FUNCTION_BLOCK FB_Station IMPLEMENTS IStation
VAR_INPUT
END_VAR
VAR_OUTPUT
END_VAR
VAR
    _Position          : REFERENCE TO FB_Position;
    _Process           : REFERENCE TO FB_AUT_ABSTRACT;
    _WaitPosOffset     : LREAL; // offset of the station position, should always be negative
    _iMaxWaitingMovers : INT;   // Maximum of waiting mover in front of the station

    _ApproachScenario : ApproachScenario_e := ApproachScenario_e.WaitOnFinishedProcess;

    _iID : INT := 0; // instance ID, is set during FB_Init using the value of _iInstanceCounter 
END_VAR
VAR_STAT
    _iInstanceCounter : INT := 1; // instance counter
END_VAR

PROPERTY ApproachScenario : ApproachScenario_e
GET
ApproachScenario := THIS^._ApproachScenario;
END_GET
SET
THIS^._ApproachScenario := ApproachScenario;
END_SET
END_PROPERTY

// Return true if the given object is equal to THIS^
METHOD Equals : BOOL
VAR_INPUT
    Station : REFERENCE TO FB_Station;
END_VAR
Equals := FALSE;

IF __ISVALIDREF(Station) THEN
    Equals := THIS = ADR(Station);
END_IF
END_METHOD

METHOD FB_init : BOOL
VAR_INPUT
    bInitRetains      : BOOL; // if TRUE, the retain variables are initialized (warm start / cold start)
    bInCopyCode       : BOOL; // if TRUE, the instance afterwards gets moved into the copy code (online change)
    Position          : REFERENCE TO FB_Position;
    Process           : REFERENCE TO FB_AUT_ABSTRACT;
    WaitPosOffset     : LREAL;
    ApproachScenario  : ApproachScenario_e;
    iMaxWaitingMovers : INT;
END_VAR
THIS^._iID               := THIS^._iInstanceCounter;
THIS^._iInstanceCounter  := THIS^._iInstanceCounter + 1;
THIS^._Position          REF= Position;
THIS^._Process           REF= Process;
THIS^._WaitPosOffset     := WaitPosOffset;
THIS^._ApproachScenario  := ApproachScenario;
THIS^._iMaxWaitingMovers := iMaxWaitingMovers;
END_METHOD

// the maxuimum number of waiting movers at the front of the station
PROPERTY iMaxWaitingMovers : INT
GET
iMaxWaitingMovers := THIS^._iMaxWaitingMovers;
END_GET
SET
THIS^._iMaxWaitingMovers := iMaxWaitingMovers;
END_SET
END_PROPERTY

PROPERTY Position : REFERENCE TO FB_Position
GET
Position REF=_Position;
END_GET
SET
_Position REF=Position;
END_SET
END_PROPERTY

PROPERTY Process : REFERENCE TO FB_AUT_ABSTRACT
GET
Process REF=_Process;
END_GET
SET
_Process REF= Process;
END_SET
END_PROPERTY

METHOD SetWaitPosOffset : REFERENCE TO FB_Station
VAR_INPUT
	WaitPosOffset : LREAL; // offset position from the given station, must be negative
END_VAR
IF _WaitPosOffset < 0 THEN
    _WaitPosOffset := WaitPos;
END_IF

SetWaitPosOffset REF= THIS^;
END_METHOD

METHOD ToString : STRING
VAR_INPUT
END_VAR
VAR
END_VAR
ToString := CONCAT('FB_Station_', TO_STRING(THIS^._iID));
END_METHOD

PROPERTY PUBLIC WaitPos : LREAL
GET
WaitPos := _WaitPosOffset + this^._Position.lrWorkPosition;
END_GET
SET
IF WaitPos < THIS^._Position.lrWorkPosition THEN
    _WaitPosOffset := WaitPos - THIS^._Position.lrWorkPosition;
END_IF
END_SET
END_PROPERTY

END_FUNCTION_BLOCK

(* stored: Version 1.1.0.1, ProductVersion 3.1.4024.6
   POU FB_Station: Id {76f3a0a5-7330-41a9-8dcd-67e3fa45891a}, SpecialFunc None
   Property ApproachScenario: Id {39b39f49-19c1-4773-90ff-7d9f9dd0bc2b}
   Get Get: Id {c7ab1366-26ac-4d26-8a07-2e23989dbdf5}
   Set Set: Id {c657ec57-92e0-4d09-9356-1fe7958f2743}
   Method Equals: Id {c76b8ece-aab6-47d5-90c3-9d4c81b08fdb}
   Method FB_init: Id {898dafd4-0828-4ee9-bb08-7822f297b3cc}
   Property iMaxWaitingMovers: Id {6a45a41f-3689-4688-9ba9-b8da1a5ddf71}
   Get Get: Id {e9a9e870-7f1d-4040-b314-a5cfa5de9a7d}
   Set Set: Id {15534dbf-4933-48be-bdb5-55a0a0a3d73e}
   Property Position: Id {b021e593-80f7-4dca-adcc-e8a0edd62ea6}
   Get Get: Id {4a41f306-d439-4214-a524-8ce6f093a989}
   Set Set: Id {062b4c53-3279-46a7-994d-891e38993d44}
   Property Process: Id {0980d319-73c1-4cb0-83fe-b31ceaca6583}
   Get Get: Id {dc489d80-96a7-40ae-a3fa-8fc50f9f2c71}
   Set Set: Id {dc717f6a-ec5a-4b69-ba84-d7f4fc9c2ad2}
   Method SetWaitPosOffset: Id {e7b8aa6e-20f0-4552-8aa4-a2e00be23ec6}
   Method ToString: Id {754f94dd-b150-4629-9617-347a61796109}
   Property WaitPos: Id {2c905c9e-5fcb-4960-a6c3-5642ee2d9ad4}
   Get Get: Id {0ad40636-1317-45d8-b399-d0cf3abd9a1b}
   Set Set: Id {3b6ab7a2-c7a0-4fee-a117-a681a2d3451b} *)
